// TIA Portal V19 export
TYPE "ValveMachine_Manager"
// stored: Access Published
   STRUCT
      EnableStopDoorOpeningReq : Bool := TRUE;
      EnableStopInPhase : Bool := TRUE;
      EnableStopProgrammed : Bool := TRUE;
      Control_ON : Bool := FALSE;
      Rest : Bool := FALSE;
      Work : Bool := FALSE;
   END_STRUCT;
END_TYPE
